FUNCTION_BLOCK ROUND_AR (* AR-Adapter-Wrapper um OSCAT ROUND - bruckt zwischen adapter und OSCAT, ohne dass eine der beiden Basisbibliotheken von der anderen abhaengt. N (Nachkommastellen) als Klartext-InputVar durchgereicht (Default 2) *)
  (* Standard: 61499-2; Description: Copyright (c) 2026 Meisterschulen am Ostbahnhof This program and the accompanying materials are made available under the terms of the Eclipse Public License 2.0 which is available at https://www.eclipse.org/legal/epl-2.0/ SPDX-License-Identifier: EPL-2.0 *)
  (* Version 1.1, 2026-09-20, Franz Höpfinger, Meisterschulen am Ostbahnhof, Bugfix: N wurde nur per plain DataConnection an ROUND durchgereicht, ausgeloest einzig ueber AR_IN.E1 - dieser Wrapper hatte ueberhaupt kein EventInput und damit keine Moeglichkeit fuer eine With-Verknuepfung (IEC 61499 - ungebundene Vars werden nicht zuverlaessig gelesen). Neues explizites REQ-EventInput ergaenzt (parallel zu AR_IN.E1, beide -> ROUND.REQ) mit With N. *)
  (* Version 1.0, 2026-09-17, Franz Höpfinger, Meisterschulen am Ostbahnhof, Initial implementation of ROUND_AR wrapper FB - E_D_FF_ANY_1 als Aenderungsfilter (EO/AR_OUT.E1 nur bei tatsaechlicher Wertaenderung), analog CTRL_PI_AR/FT_DERIV_AR in diesem Projekt *)
  PACKAGE OSCAT_adapter::Mathematical;
  (* Documentation:
  ROUND_AR
   🇩🇪 Deutsch
   AR-Adapter-Wrapper um OSCAT::Basic::POUs::Mathematical::ROUND (rundet in auf N Nachkommastellen, 0 bis 8 Stellen). N ist als Klartext-InputVar (Default 2) deklariert. Ein explizites REQ-EventInput (mit With N) erlaubt den manuellen/periodischen Aufruf zusaetzlich zum automatischen Ausloesen ueber AR_IN.E1 (IEC 61499 - With-Verknuepfung fuer zuverlaessiges Einlesen der Parameter).
   Reine Adapter-Grenze
    - AR_IN (Socket, AR): Eingangssignal (REAL)
   - AR_OUT (Plug, AR): gerundetes Ergebnis (REAL)
    E_D_FF_ANY_1 (Standardbibliothek events-3.0.0) filtert Aenderungen: AR_OUT.E1 feuert nur, wenn sich das gerundete Ergebnis seit dem letzten Aufruf tatsaechlich geaendert hat - gleiches Muster wie bei den bestehenden FT_DERIV_AR/CTRL_PI_AR-Wrappern in diesem Projekt (dort mit E_D_FF_ANY_3/_4 fuer mehrere Werte gleichzeitig).
   Warum ein eigener Wrapper?
   ROUND ist eine reine OSCAT-Function ohne Adapter-Schnittstelle. adapter soll nicht von OSCAT abhaengen (und umgekehrt) - die Bruecke liegt daher in diesem dritten Bibliotheksprojekt (OSCAT_adapter), das von beiden abhaengt.
   🇬🇧 English
   AR-adapter wrapper around OSCAT::Basic::POUs::Mathematical::ROUND (rounds in to N decimal places, 0 to 8 digits). N is a plain InputVar (default 2). An explicit REQ event input (with With N binding) enables manual or periodic execution in addition to automatic triggering via AR_IN.E1 (per IEC 61499, binding input variables via With for reliable reading).
   Pure adapter boundary
    - AR_IN (socket, AR): input signal (REAL)
   - AR_OUT (plug, AR): rounded result (REAL)
    E_D_FF_ANY_1 (standard library events-3.0.0) filters changes: AR_OUT.E1 only fires when the rounded result actually changed since the last call - same pattern as the existing FT_DERIV_AR/CTRL_PI_AR wrappers in this project (there using E_D_FF_ANY_3/_4 for several values at once).
  *)
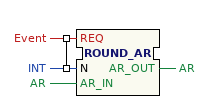
  EVENT_INPUT
    REQ WITH N; (* Explizite Ausfuehrungsanforderung (durchgereicht an ROUND.REQ, zusaetzlich zu AR_IN.E1) *)
  END_EVENT
  VAR_INPUT
    N : INT := 2; (* Nachkommastellen (durchgereicht an ROUND.N) - Platzhalter-Default 2, keine funktionale Vorgabe, per Parameter ueberschreibbar *)
  END_VAR
  SOCKETS
    AR_IN : adapter::types::unidirectional::AR; (* Eingangssignal (REAL) *)
  END_SOCKETS
  PLUGS
    AR_OUT : adapter::types::unidirectional::AR; (* Auf N Nachkommastellen gerundeter Wert (REAL) *)
  END_PLUGS
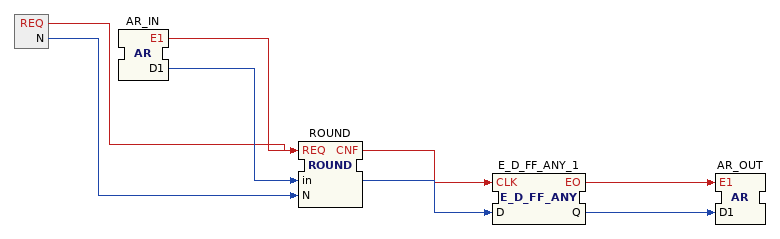
  FBS
    ROUND : OSCAT::Basic::POUs::Mathematical::ROUND;
    E_D_FF_ANY_1 : iec61499::events::E_D_FF_ANY;
  END_FBS
  EVENT_CONNECTIONS
    AR_IN.E1 TO ROUND.REQ;
    REQ TO ROUND.REQ;
    ROUND.CNF TO E_D_FF_ANY_1.CLK;
    E_D_FF_ANY_1.EO TO AR_OUT.E1;
  END_CONNECTIONS
  DATA_CONNECTIONS
    AR_IN.D1 TO ROUND.in;
    N TO ROUND.N;
    ROUND. TO E_D_FF_ANY_1.D;
    E_D_FF_ANY_1.Q TO AR_OUT.D1;
  END_CONNECTIONS
END_FUNCTION_BLOCK
